TYPE SValue :
STRUCT
	DataType: EDataType;
	Value: UValues;
	Defined: BOOL;
END_STRUCT
END_TYPE

(* stored: Version 1.1.0.1
   DUT SValue: Id {8b32d60a-f461-44ec-8937-d4b17922f5fb} *)
